// TIA Portal V17 export
// export: Created 2024-09-02T12:50:07.5499668Z, ExportSetting WithDefaults, DisplayName Totally Integrated Automation Portal, DisplayVersion V17, DisplayName TIA Portal Openness, DisplayVersion V17, DisplayName TIA Portal Version Control Interface, DisplayVersion V17, DisplayName STEP 7 Professional, DisplayVersion V17, DisplayName STEP 7 Safety, DisplayVersion V17, DisplayName WinCC Professional, DisplayVersion V17
DATA_BLOCK "GraDB1_FG01_Transport_OP70"   // DB1261
{ S7_Optimized_Access := 'TRUE'; DB_Accessible_From_OPC_UA := 'FALSE' }
AUTHOR : VAF
FAMILY : SK
NAME : SK
VERSION : 0.1
// stored: AutoNumber false, DBAccessibleFromOPCUA false, IsOnlyStoredInLoadMemory false, IsRetainMemResEnabled false, IsWriteProtectedInAS false, MemoryReserve 0
   VAR
      Home { ExternalWritable := 'False'} : Bool;   // Grundstellung / Homeposition
      Home_Mechanic { ExternalWritable := 'False'} : Bool;   // Grundstellung Mechanik / Basic position mechanic
      Home_SQ { ExternalWritable := 'False'} : Bool;   // Grundstellung Schrittkette / Basic position Step chain
      Finished_Reset_PreStp { ExternalWritable := 'False'} : Bool;   // Fertigmeldung Ablöschen Vorstopper / Finish message Delete Prestopper
      Finished_Reset_Stp { ExternalWritable := 'False'} : Bool;   // Fertigmeldung Ablöschen Stopper / Finish message Delete Stopper
      Entry_Permit_ON_Stopper { ExternalWritable := 'False'} : Bool;   // Freigabe Einlauf / Enable inlet
      Wait_For_Pallet { ExternalWritable := 'False'} : Bool;   // Warte auf WT in Station / Wait for Pallet in Station
      Pallet_Leaving_Prestopper { ExternalWritable := 'False'} : Bool;   // WT ist ausgelaufen Vorstopper / Pallet has run out Vorstopper
      Pallet_Leaving_Stopper { ExternalWritable := 'False'} : Bool;   // WT ist ausgelaufen Stopper / Pallet has run out Stopper
      Swk_Leaving_PreStp { ExternalWritable := 'False'} : Bool;   // Kontrolle Auslauf Vorstopper / Control spout pre-stopper
      Swk_Leaving_Stp { ExternalWritable := 'False'} : Bool;   // Kontrolle Auslauf Stopper / Control spout stopper
      Swk_Rotate_Table_PreStp { ExternalWritable := 'False'} : Bool;   // Kontrolle Drehteller Vorstopper / Control turntable pre-stopper
      Swk_Rotate_Table_Stp { ExternalWritable := 'False'} : Bool;   // Kontrolle Drehteller Stopper / Control turntable stopper
      Swk_Traffic_Sensor { ExternalWritable := 'False'} : Bool;   // Kontrolle Stauabfrage / Control congestion check
      Pallet_In_Station { ExternalWritable := 'False'} : Bool;   // WT in Station vorhanden / Pallet available in station
   END_VAR
   VAR RETAIN
      Finished : Bool := false;   // Fertigmeldung / Finished message
      Moby_Reading_Done_PreStp : Bool;   // MOBY1: Auswertung Fertig / MOBY1: Evaluation finished
      Moby_Saveing_Done_PreStp : Bool;   // MOBY1: Rückberechnung Fertig / MOBY1: Saving Finished
      Moby_Reading_Done_Stp : Bool;   // MOBY1: Auswertung Fertig / MOBY1: Evaluation finished
      Moby_Saveing_Done_Stp : Bool;   // MOBY1: Rückberechnung Fertig / MOBY1: Saving Finished
      With_Processing : Bool;   // MOBY: Station mit Bearbeitung / MOBY: Station with machining
      Without_Processing : Bool;   // MOBY: Station ohne Bearbeitung / MOBY: Station with machining
      Release_BEA_1 : Bool;   // Bearbeitungsfreigabe BEA 1 / Processing enable BEA1
      Release_BEA_2 : Bool;   // Bearbeitungsfreigabe BEA 2 / Processing enable BEA2
      Release_BEA_3 : Bool;   // Bearbeitungsfreigabe BEA 3 / Processing enable BEA3
      Release_BEA_4 : Bool;   // Bearbeitungsfreigabe BEA 4 / Processing enable BEA4
      Release_BEA_5 : Bool;   // Bearbeitungsfreigabe BEA 5 / Processing enable BEA5
      Release_BEA_6 : Bool;   // Bearbeitungsfreigabe BEA 6 / Processing enable BEA6
      Release_BEA_7 : Bool;   // Bearbeitungsfreigabe BEA 7 / Processing enable BEA7
      Release_BEA_8 : Bool;   // Bearbeitungsfreigabe BEA 8 / Processing enable BEA8
   END_VAR
   VAR
      Release_Sequences_BEA { S7_SetPoint := 'True'} : "TypeSKS";   // Schrittmerker / Step marker
      Part_Counter_Stopper { S7_SetPoint := 'True'} : "TypeSKS_COUNTER";   // Schrittmerker / Step marker
      conveyors { S7_SetPoint := 'True'} : "TypeSKS_MOTOR";   // Schrittmerker / Step marker
      SLG1 { S7_SetPoint := 'True'} : "TypeSKS_SLG";   // Schrittmerker / Step marker
      "MM10 Prestopper" { S7_SetPoint := 'True'} : "TypeSKS_STP";   // Schrittmerker / Step marker
      "MM20 Stopper" { S7_SetPoint := 'True'} : "TypeSKS_STP";   // Schrittmerker / Step marker
      "MM30/31 Index" { S7_SetPoint := 'True'} : "TypeSKS_VERT";   // Schrittmerker / Step marker
      Tracebility_off { S7_SetPoint := 'True'} : Bool;
   END_VAR
BEGIN
END_DATA_BLOCK
